FUNCTION_BLOCK EncoderSignalProcessor
VAR_INPUT
	pulseA : BOOL;
	pulseB : BOOL;
	//reset :	
	referencePositionSensor : BOOL;
	referencePosition: INT := 0;
END_VAR
VAR_OUTPUT
	direction : BOOL;
	position : INT;
END_VAR
VAR
	trigger : BOOL;
	direction_ : BOOL;
	count_ : INT;
	
END_VAR
VAR // added by the converter: edge detectors and wires of the graphical bodies
    _rt1, _rt2, _rt3, _rt4 : R_TRIG;
    _ft1, _ft2, _ft3, _ft4 : F_TRIG;
END_VAR

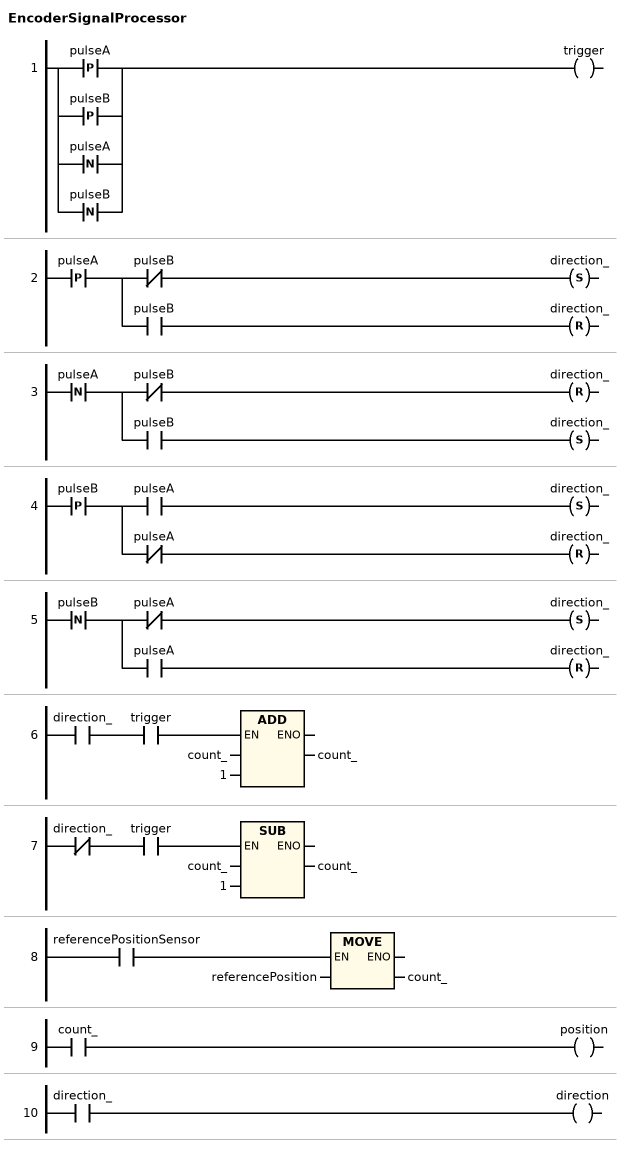
// NETWORK 1
_rt1(CLK := pulseA);
_rt2(CLK := pulseB);
_ft1(CLK := pulseA);
_ft2(CLK := pulseB);
trigger := _rt1.Q OR _rt2.Q OR _ft1.Q OR _ft2.Q;

// NETWORK 2
_rt3(CLK := pulseA);
direction_ S= _rt3.Q AND NOT pulseB;
direction_ R= _rt3.Q AND pulseB;

// NETWORK 3
_ft3(CLK := pulseA);
direction_ R= _ft3.Q AND NOT pulseB;
direction_ S= _ft3.Q AND pulseB;

// NETWORK 4
_rt4(CLK := pulseB);
direction_ S= _rt4.Q AND pulseA;
direction_ R= _rt4.Q AND NOT pulseA;

// NETWORK 5
_ft4(CLK := pulseB);
direction_ S= _ft4.Q AND NOT pulseA;
direction_ R= _ft4.Q AND pulseA;

// NETWORK 6
IF direction_ AND trigger THEN count_ := count_ + 1; END_IF

// NETWORK 7
IF NOT direction_ AND trigger THEN count_ := count_ - 1; END_IF

// NETWORK 8
IF referencePositionSensor THEN count_ := referencePosition; END_IF

// NETWORK 9
position := count_;

// NETWORK 10
direction := direction_;

END_FUNCTION_BLOCK

(* stored: Version 1.1.0.1, ProductVersion 3.1.4024.12
   POU EncoderSignalProcessor: Id {3bfd9821-10a4-4c0c-8aa4-82b71e8ea22a}, SpecialFunc None *)
